FUNCTION_BLOCK UR3_StateMachine

VAR_INPUT
	init_: BOOL:= FALSE;
	G_STATE: INT:=-1;

END_VAR


VAR
	//internal aux state
	I_STATE : INT:=-1;
END_VAR


VAR_OUTPUT
	State_complete : BOOL:= FALSE;
	Act_Gl_State :INT:=-1;
	Act_In_State: INT:=-1;
END_VAR

VAR CONSTANT 
	

	
END_VAR

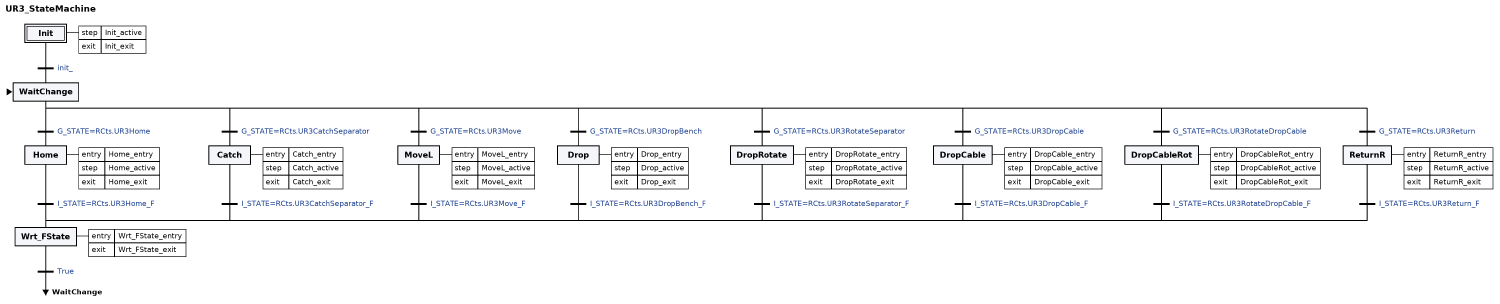
INITIAL_STEP Init:
    Init_active(N);  // step action
    Init_exit(P0);  // exit action
END_STEP
TRANSITION FROM Init TO WaitChange
    := init_;
END_TRANSITION
STEP WaitChange:
END_STEP
TRANSITION FROM WaitChange TO Home
    := G_STATE=RCts.UR3Home;
END_TRANSITION
STEP Home:
    Home_entry(P1);  // entry action
    Home_active(N);  // step action
    Home_exit(P0);  // exit action
END_STEP
TRANSITION FROM Home TO Wrt_FState
    := I_STATE=RCts.UR3Home_F;
END_TRANSITION
TRANSITION FROM WaitChange TO Catch
    := G_STATE=RCts.UR3CatchSeparator;
END_TRANSITION
STEP Catch:
    Catch_entry(P1);  // entry action
    Catch_active(N);  // step action
    Catch_exit(P0);  // exit action
END_STEP
TRANSITION FROM Catch TO Wrt_FState
    := I_STATE=RCts.UR3CatchSeparator_F;
END_TRANSITION
TRANSITION FROM WaitChange TO MoveL
    := G_STATE=RCts.UR3Move;
END_TRANSITION
STEP MoveL:
    MoveL_entry(P1);  // entry action
    MoveL_active(N);  // step action
    MoveL_exit(P0);  // exit action
END_STEP
TRANSITION FROM MoveL TO Wrt_FState
    := I_STATE=RCts.UR3Move_F;
END_TRANSITION
TRANSITION FROM WaitChange TO Drop
    := G_STATE=RCts.UR3DropBench;
END_TRANSITION
STEP Drop:
    Drop_entry(P1);  // entry action
    Drop_active(N);  // step action
    Drop_exit(P0);  // exit action
END_STEP
TRANSITION FROM Drop TO Wrt_FState
    := I_STATE=RCts.UR3DropBench_F;
END_TRANSITION
TRANSITION FROM WaitChange TO DropRotate
    := G_STATE=RCts.UR3RotateSeparator;
END_TRANSITION
STEP DropRotate:
    DropRotate_entry(P1);  // entry action
    DropRotate_active(N);  // step action
    DropRotate_exit(P0);  // exit action
END_STEP
TRANSITION FROM DropRotate TO Wrt_FState
    := I_STATE=RCts.UR3RotateSeparator_F;
END_TRANSITION
TRANSITION FROM WaitChange TO DropCable
    := G_STATE=RCts.UR3DropCable;
END_TRANSITION
STEP DropCable:
    DropCable_entry(P1);  // entry action
    DropCable_active(N);  // step action
    DropCable_exit(P0);  // exit action
END_STEP
TRANSITION FROM DropCable TO Wrt_FState
    := I_STATE=RCts.UR3DropCable_F;
END_TRANSITION
TRANSITION FROM WaitChange TO DropCableRot
    := G_STATE=RCts.UR3RotateDropCable;
END_TRANSITION
STEP DropCableRot:
    DropCableRot_entry(P1);  // entry action
    DropCableRot_active(N);  // step action
    DropCableRot_exit(P0);  // exit action
END_STEP
TRANSITION FROM DropCableRot TO Wrt_FState
    := I_STATE=RCts.UR3RotateDropCable_F;
END_TRANSITION
TRANSITION FROM WaitChange TO ReturnR
    := G_STATE=RCts.UR3Return;
END_TRANSITION
STEP ReturnR:
    ReturnR_entry(P1);  // entry action
    ReturnR_active(N);  // step action
    ReturnR_exit(P0);  // exit action
END_STEP
TRANSITION FROM ReturnR TO Wrt_FState
    := I_STATE=RCts.UR3Return_F;
END_TRANSITION
STEP Wrt_FState:
    Wrt_FState_entry(P1);  // entry action
    Wrt_FState_exit(P0);  // exit action
END_STEP
TRANSITION FROM Wrt_FState TO WaitChange
    := True;
END_TRANSITION

ACTION Catch_active:
//read register from robot and chek is can read 2 or more correct values 
IF ck_state(RCts.UR3,RCts.UR3CatchSeparator_I) THEN
	 I_STATE:= RCts.UR3CatchSeparator_I;
ELSIF ck_state(RCts.UR3,RCts.UR3CatchSeparator_F) THEN
	I_STATE := RCts.UR3CatchSeparator_F;
END_IF

//read internal variable and write over output variable
Act_In_State := I_STATE;
END_ACTION

ACTION Catch_entry:
//write state variables to robot, to execute respective state.
wr_state(RCts.UR3,RCts.UR3CatchSeparator);
//write the retain state variable 
Act_Gl_State:=RCts.UR3CatchSeparator;
END_ACTION

ACTION Catch_exit:
//write reset state variables to robot.
wr_state(RCts.UR3,RCts.RESET_STATE);
//reset Global state variable
G_STATE := -1;
END_ACTION

ACTION Drop_active:
//read register from robot and chek is can read 2 or more correct values 
IF ck_state(RCts.UR3,RCts.UR3DropBench_I) THEN
	 I_STATE:= RCts.UR3DropBench_I;
ELSIF ck_state(RCts.UR3,RCts.UR3DropBench_F) THEN
	I_STATE := RCts.UR3DropBench_F;
END_IF


//read internal variable and write over output variable
Act_In_State := I_STATE;
END_ACTION

ACTION Drop_entry:
//write state variables to robot, to execute respective state.
wr_state(RCts.UR3,RCts.UR3DropBench);
//write the retain state variable 
Act_Gl_State:=RCts.UR3DropBench;
END_ACTION

ACTION Drop_exit:
//write reset state variables to robot.
wr_state(RCts.UR3,RCts.RESET_STATE);
//Assign a value according to the variable UserState
//-1 or respective NEXT state  CS.UR3DropBench
//wr_GL_STATE(CS.UR5Camera1,UserState);

//reset Global state variable
G_STATE := -1;
END_ACTION

ACTION DropCable_active:
//read register from robot and chek is can read 2 or more correct values 
IF ck_state(RCts.UR3,RCts.UR3DropCable_I) THEN
	 I_STATE:= RCts.UR3DropCable_I;
ELSIF ck_state(RCts.UR3,RCts.UR3DropCable_F) THEN
	I_STATE := RCts.UR3DropCable_F;
END_IF

//read internal variable and write over output variable
Act_In_State := I_STATE;
END_ACTION

ACTION DropCable_entry:
//write state variables to robot, to execute respective state.
wr_state(RCts.UR3,RCts.UR3DropCable);
//write the retain state variable 
Act_Gl_State:=RCts.UR3DropCable;
END_ACTION

ACTION DropCable_exit:
//write reset state variables to robot.
wr_state(RCts.UR3,RCts.RESET_STATE);
//reset Global state variable
G_STATE := -1;
END_ACTION

ACTION DropCableRot_active:
//read register from robot and chek is can read 2 or more correct values 
IF ck_state(RCts.UR3,RCts.UR3RotateDropCable_I) THEN
	 I_STATE:= RCts.UR3RotateDropCable_I;
ELSIF ck_state(RCts.UR3,RCts.UR3RotateDropCable_F) THEN
	I_STATE := RCts.UR3RotateDropCable_F;
END_IF


//read internal variable and write over output variable
Act_In_State := I_STATE;
END_ACTION

ACTION DropCableRot_entry:
//write state variables to robot, to execute respective state.
wr_state(RCts.UR3,RCts.UR3RotateDropCable);
//write the retain state variable 
Act_Gl_State:=RCts.UR3RotateDropCable;
END_ACTION

ACTION DropCableRot_exit:
//write reset state variables to robot.
wr_state(RCts.UR3,RCts.RESET_STATE);
//reset Global state variable
G_STATE := -1;
END_ACTION

ACTION DropRotate_active:

//read register from robot and chek is can read 2 or more correct values 
IF ck_state(RCts.UR3,RCts.UR3RotateSeparator_I) THEN
	 I_STATE:= RCts.UR3RotateSeparator_I;
ELSIF ck_state(RCts.UR3,RCts.UR3RotateSeparator_F) THEN
	I_STATE := RCts.UR3RotateSeparator_F;
END_IF

//read internal variable and write over output variable
Act_In_State := I_STATE;
END_ACTION

ACTION DropRotate_entry:
//write state variables to robot, to execute respective state.
wr_state(RCts.UR3,RCts.UR3RotateSeparator);
//write the retain state variable 
Act_Gl_State:=RCts.UR3RotateSeparator;
END_ACTION

ACTION DropRotate_exit:
//write reset state variables to robot.
wr_state(RCts.UR3,RCts.RESET_STATE);
//reset Global state variable
G_STATE := -1;
END_ACTION

ACTION Home_active:
//read register from robot and chek is can read 2 or more correct values 
IF ck_state(RCts.UR3,RCts.UR3Home_I) THEN
	 I_STATE:= RCts.UR3Home_I;
ELSIF ck_state(RCts.UR3,RCts.UR3Home_F) THEN
	I_STATE := RCts.UR3Home_F;
END_IF

//read internal variable and write over output variable
Act_In_State := I_STATE;
END_ACTION

ACTION Home_entry:
//write state variables to robot, to execute respective state.
wr_state(RCts.UR3,RCts.UR3Home);
//write the retain state variable 
Act_Gl_State:=RCts.UR3Home;
END_ACTION

ACTION Home_exit:
//write reset state variables to robot.
wr_state(RCts.UR3,RCts.RESET_STATE);
//reset Global state variable
G_STATE := -1;
END_ACTION

ACTION Init_active:

END_ACTION

ACTION Init_exit:
//write reset state variables to robot.
wr_state(RCts.UR3,RCts.RESET_STATE);
//write reset state variables to robot.
//wr_state(CS.UR5,RESET_STATE);
END_ACTION

ACTION MoveL_active:
//read register from robot and chek is can read 2 or more correct values 
IF ck_state(RCts.UR3,RCts.UR3Move_I) THEN
	 I_STATE:= RCts.UR3Move_I;
ELSIF ck_state(RCts.UR3,RCts.UR3Move_F) THEN
	I_STATE := RCts.UR3Move_F;
END_IF


//read internal variable and write over output variable
Act_In_State := I_STATE;
END_ACTION

ACTION MoveL_entry:
//write state variables to robot, to execute respective state.
wr_state(RCts.UR3,RCts.UR3Move);
//write the retain state variable 
Act_Gl_State:=RCts.UR3Move;
END_ACTION

ACTION MoveL_exit:
//write reset state variables to robot.
wr_state(RCts.UR3,RCts.RESET_STATE);
//reset Global state variable
G_STATE := -1;
END_ACTION

ACTION ReturnR_active:
//read register from robot and chek is can read 2 or more correct values 
IF ck_state(RCts.UR3,RCts.UR3Return_I) THEN
	 I_STATE:= RCts.UR3Return_I;
ELSIF ck_state(RCts.UR3,RCts.UR3Return_F) THEN
	I_STATE := RCts.UR3Return_F;
END_IF

//read internal variable and write over output variable
Act_In_State := I_STATE;
END_ACTION

ACTION ReturnR_entry:
//write state variables to robot, to execute respective state.
wr_state(RCts.UR3,RCts.UR3Return);
//write the retain state variable 
Act_Gl_State:=RCts.UR3Return;
END_ACTION

ACTION ReturnR_exit:
//write reset state variables to robot.
wr_state(RCts.UR3,RCts.RESET_STATE);
//reset Global state variable
G_STATE := -1;
END_ACTION

ACTION UR3Move_entry:
//write state variables to robot, to execute respective state.
wr_state(RCts.UR3,RCts.UR3CatchSeparator);
//write the retain state variable 
Act_Gl_State:=RCts.UR3CatchSeparator;
END_ACTION

ACTION UR3Move_exit:
//write reset state variables to robot.
wr_state(RCts.UR3,RCts.RESET_STATE);
//reset Global state variable
G_STATE := -1;
END_ACTION

ACTION Wrt_FState_entry:
//write output variable to indicate that the robot execute the state 
State_complete := TRUE;
END_ACTION

ACTION Wrt_FState_exit:
//write output variable to indicate that the robot execute the state 
State_complete := FALSE;
init_:=FALSE;

G_STATE := -1;
//rest internat state variable
I_STATE :=-1;
END_ACTION

END_FUNCTION_BLOCK

(* stored: Version 1.1.0.1, ProductVersion 3.1.4024.4
   POU UR3_StateMachine: Id {8ccd1054-69f9-4e2e-9068-25c51f0ebb46}, SpecialFunc None
   Action Catch_active: Id {dee5f8fb-cc74-4020-9f02-a479e851a7c5}
   Action Catch_entry: Id {eb0e7c9a-2688-461c-9fcf-73e6bb2707a7}
   Action Catch_exit: Id {1839f270-85e5-4e93-a2e6-bfc34edc9417}
   Action Drop_active: Id {6c2d05ba-c789-4677-9343-33bbed149cdf}
   Action Drop_entry: Id {3f67d0c1-a53c-4a21-8e64-84fbcea3f2b2}
   Action Drop_exit: Id {58c43fbe-b196-442e-a973-b1633ddf2aa1}
   Action DropCable_active: Id {3d87289e-ce57-4bca-80af-0e5162b89757}
   Action DropCable_entry: Id {a7ebd044-5109-4224-87e6-993b8d1f4ca4}
   Action DropCable_exit: Id {28b49d7a-1073-4215-a5e9-2c5ae70bc743}
   Action DropCableRot_active: Id {e839c00b-168d-4c6a-823f-92517fdd4c6e}
   Action DropCableRot_entry: Id {62ad4158-aeef-4e82-bb7a-1ec2f064e009}
   Action DropCableRot_exit: Id {55ac6059-1b6d-4c36-b0f4-2f9ed5380db5}
   Action DropRotate_active: Id {e2df560a-e202-42ab-94cf-374c2c515e2a}
   Action DropRotate_entry: Id {a7d14bfd-688a-4821-9548-5d0f26f49ac8}
   Action DropRotate_exit: Id {62a7f7c3-fa4c-4c2d-a174-81f106cdf371}
   Action Home_active: Id {86a7559d-df27-4823-b7d8-8387dec4121e}
   Action Home_entry: Id {4b6ffa9b-16e0-4651-8086-b1f5bb37d863}
   Action Home_exit: Id {030f12c3-7881-44f6-8d96-c86ed2b5cf69}
   Action Init_active: Id {440cb59c-cdf4-4a4c-a127-f3d5384a7bcc}
   Action Init_exit: Id {14731561-fb27-43fc-9de4-1299a05bea9f}
   Action MoveL_active: Id {1b445c3c-da20-4309-a5da-1ee9f9fceade}
   Action MoveL_entry: Id {4e17fb59-0a23-4c16-adfa-b260e4452a74}
   Action MoveL_exit: Id {a2269d4d-fce5-446a-9271-0fba53b85dfb}
   Action ReturnR_active: Id {4f2fbd99-2c40-4660-ab3d-ec9c0eaf73e5}
   Action ReturnR_entry: Id {913078bb-7137-4955-934c-f46f467ab1d3}
   Action ReturnR_exit: Id {87f97ffe-9cfe-45c7-b5ba-940214f29c90}
   Action UR3Move_entry: Id {e7cdf7ef-6cdb-4396-b0be-dba08508b264}
   Action UR3Move_exit: Id {39c19447-93c3-426a-876f-b3cc3df54043}
   Action Wrt_FState_entry: Id {7b07250d-74d7-4bf9-bfb1-e861ae9e0656}
   Action Wrt_FState_exit: Id {d70e1a24-d99f-43db-b5ce-f45000f7b01b} *)
